(* IEC 61131-3 sources: AXOpen/src/components.rexroth.drives/ctrl/src/AxoIndraDrive (part 3) *)

            Valid			:= 	MC_ReadParameterDone_;
            Busy			:= 	MC_ReadParameterActive_;
            Error			:= 	MC_ReadParameterError_;
            ErrorID			:= 	TO_DINT(MC_ReadParameterErrorID_);
            IF Valid THEN
                Value			:= 	MC_ReadParameterValue_;
            ELSE
                Value			:= 	0;
            END_IF;
        END_METHOD

        ///<summary>
        /// This method returns the value of a vendor specific parameter with datatype REAL.
        ///<summary>
        VAR INTERNAL
            MC_ReadRealParameterEnable_PV		: 	BOOL := FALSE;		//Enable - previous value
            MC_ReadRealParameterDone_PV			:	BOOL := FALSE;		//Done - previous value
            MC_ReadRealParameterCallNumber		: 	INT; 				//Call number of the method MC_ReadRealParameter
            MC_ReadRealParameterNumber_PV		: 	DINT;				//ParameterNumber - previous value (stored at rising edge of the Enable)
            MC_ReadRealParameterFirstCall		: 	BOOL;				//First call of the method MC_ReadRealParameter
            MC_ReadRealParameterDone_			:	BOOL;
            MC_ReadRealParameterActive_			:	BOOL := FALSE;
            MC_ReadRealParameterError_			:	BOOL;
            MC_ReadRealParameterErrorID_		:	eAxoIndraDriveErrorCode;
            MC_ReadRealParameterValue_			:	REAL;
        END_VAR
        METHOD PUBLIC OVERRIDE MC_ReadRealParameter
            VAR_INPUT
                AxisRef         :   AXOpen.Components.Abstractions.Drives.IAxoAxisReference;
                Enable          :   BOOL;                       //  Get the value of the parameter continuously while enabled
                ParameterNumber :   DINT;                       //  Number of the parameter. One can also use symbolic parameter names which are declared as VAR CONST.
            END_VAR
            VAR_OUTPUT
                Valid           :   BOOL;                       //  A valid output is available at the method
                Busy            :   BOOL;                       //  The method is not finished and new output values are to be expected
                Error           :   BOOL;                       //  Signals that an error has occurred within the method
                ErrorID         :   DINT;                       //  Error identification
                Value           :   REAL;                       //  Value of the specified parameter in the datatype, as specified by the vendor
            END_VAR
            VAR
                _AxisReference :  REF_TO AXOpen.Components.Rexroth.Drives.AxoIndraDriveAxisReference;
                Dummy : BOOL;
            END_VAR

            _AxisReference ?= AxisRef;

            Messenger.ActivateOnCondition(ULINT#1413,_AxisReference = NULL, eAxoMessageCategory#ProgrammingError);

            IF(_AxisReference = NULL) THEN
                RETURN;
            END_IF;

            IF Enable THEN
                MC_ReadRealParameterFirstCall := TRUE;
                IF _AxisReference^.Data.CheckAccessOK THEN
                    IF Enable AND NOT MC_ReadRealParameterEnable_PV THEN(*	raising edge of Enable *)
                        IF NOT _AxisReference^.Data.ActiveAcyclicCommunication THEN
                            _AxisReference^.Data.CallNumberAcyclic := _AxisReference^.Data.CallNumberAcyclic + INT#2;
                            MC_ReadRealParameterCallNumber := _AxisReference^.Data.CallNumberAcyclic;
                            MC_ReadRealParameterNumber_PV := ParameterNumber;
                            _AxisReference^.Data.WriteParameter := FALSE;
                            _AxisReference^.Data.SelectDataType := UINT#2;
                            _AxisReference^.Data.ParameterNumber := MC_ReadRealParameterNumber_PV;
                            MC_ReadRealParameterError_ := FALSE;
                            MC_ReadRealParameterErrorID_ := AXOpen.Components.Rexroth.Drives.eAxoIndraDriveErrorCode#NONE_ERROR;
                        ELSE
                            MC_ReadRealParameterError_ := TRUE;
                            MC_ReadRealParameterErrorID_ := AXOpen.Components.Rexroth.Drives.eAxoIndraDriveErrorCode#ACCESS_ERROR;
                        END_IF;
                    END_IF;
                ELSE
                    MC_ReadRealParameterCallNumber := MC_ReadRealParameterCallNumber - INT#1;
                    MC_ReadRealParameterError_ := TRUE;
                    MC_ReadRealParameterErrorID_ := AXOpen.Components.Rexroth.Drives.eAxoIndraDriveErrorCode#RESOURCE_ERROR;
                END_IF;
            END_IF;
            IF MC_ReadRealParameterFirstCall THEN
                IF MC_ReadRealParameterCallNumber = _AxisReference^.Data.CallNumberAcyclic AND Enable	THEN
                    _AxisReference^.Data.CallAxisParameterMethod := TRUE;
                    _AxisReference^.Data.EnableAcyclicCommunication := TRUE;
                    THIS.AcyclicCommunicationCall(AxisRef :=  _AxisReference , DPV1ParameterNumber := TRUE, Active => Dummy);
                    Busy := _AxisReference^.Data.ActiveAcyclicCommunication;
                    IF _AxisReference^.Data.DoneAcyclicCommunication THEN
                        MC_ReadRealParameterDone_ := TRUE;
                        MC_ReadRealParameterActive_ := FALSE;
                        MC_ReadRealParameterValue_ := _AxisReference^.Data.ReadValueReal;
                    END_IF;
                    IF _AxisReference^.Data.Error_AcyclicCommunication THEN
                        MC_ReadRealParameterCallNumber := MC_ReadRealParameterCallNumber - INT#1;
                        MC_ReadRealParameterDone_ := FALSE;
                        MC_ReadRealParameterActive_ := FALSE;
                        MC_ReadRealParameterError_ := _AxisReference^.Data.Error_AcyclicCommunication;
                        MC_ReadRealParameterErrorID_ := _AxisReference^.Data.ErrorID_AcyclicCommunication;
                        _AxisReference^.Data.CallAxisParameterMethod := TRUE;
                        _AxisReference^.Data.EnableAcyclicCommunication := FALSE;
                        THIS.AcyclicCommunicationCall(AxisRef :=  _AxisReference , DPV1ParameterNumber := TRUE, Active => Dummy);
                    ELSIF  _AxisReference^.Data.CallAxisParameterMethod THEN
                        MC_ReadRealParameterCallNumber := MC_ReadRealParameterCallNumber - INT#1;
                        MC_ReadRealParameterDone_ := FALSE;
                        MC_ReadRealParameterActive_ := FALSE;
                        MC_ReadRealParameterError_ := TRUE;
                        MC_ReadRealParameterErrorID_ := AXOpen.Components.Rexroth.Drives.eAxoIndraDriveErrorCode#RESOURCE_ERROR;
                        _AxisReference^.Data.EnableAcyclicCommunication := FALSE;
                    END_IF;
                ELSIF Enable AND MC_ReadRealParameterEnable_PV AND MC_ReadRealParameterCallNumber = _AxisReference^.Data.CallNumberAcyclic THEN
                    _AxisReference^.Data.CallAxisParameterMethod := TRUE;
                    _AxisReference^.Data.EnableAcyclicCommunication := FALSE;
                    THIS.AcyclicCommunicationCall(AxisRef :=  _AxisReference , DPV1ParameterNumber := TRUE, Active => Dummy);
                    MC_ReadRealParameterDone_ := FALSE;
                    MC_ReadRealParameterActive_ := FALSE;
                    MC_ReadRealParameterValue_ := 0;
                    MC_ReadRealParameterError_ := FALSE;
                    MC_ReadRealParameterErrorID_ := AXOpen.Components.Rexroth.Drives.eAxoIndraDriveErrorCode#NONE_ERROR;
                ELSIF NOT Enable AND MC_ReadRealParameterEnable_PV THEN
                    MC_ReadRealParameterDone_ := FALSE;
                    MC_ReadRealParameterActive_ := FALSE;
                    MC_ReadRealParameterValue_ := 0;
                    MC_ReadRealParameterError_ := FALSE;
                    MC_ReadRealParameterErrorID_ := AXOpen.Components.Rexroth.Drives.eAxoIndraDriveErrorCode#NONE_ERROR;
                    _AxisReference^.Data.ActiveAcyclicCommunication := FALSE;
                    _AxisReference^.Data.DoneAcyclicCommunication := FALSE;
                END_IF;
            END_IF;
            MC_ReadRealParameterEnable_PV := Enable;

            Valid			:= 	MC_ReadRealParameterDone_;
            Busy			:= 	MC_ReadRealParameterActive_;
            Error			:= 	MC_ReadRealParameterError_;
            ErrorID			:= 	TO_DINT(MC_ReadRealParameterErrorID_);
            IF Valid THEN
                Value			:= 	MC_ReadRealParameterValue_;
            ELSE
                Value			:= 	0;
            END_IF;
        END_METHOD

        ///<summary>
        /// This method returns the value of a vendor specific parameter with datatype BOOL.
        ///<summary>
        METHOD PUBLIC OVERRIDE MC_ReadBoolParameter
            VAR_INPUT
                AxisRef         :   AXOpen.Components.Abstractions.Drives.IAxoAxisReference;
                Enable          :   BOOL;                       //  Get the value of the parameter continuously while enabled
                ParameterNumber :   DINT;                       //  Number of the parameter. One can also use symbolic parameter names which are declared as VAR CONST.
            END_VAR
            VAR_OUTPUT
                Valid           :   BOOL;                       //  A valid output is available at the method
                Busy            :   BOOL;                       //  The method is not finished and new output values are to be expected
                Error           :   BOOL;                       //  Signals that an error has occurred within the method
                ErrorID         :   DINT;                       //  Error identification
                Value           :   BOOL;                       //  Value of the specified parameter in the datatype, as specified by the vendor
            END_VAR
            VAR
                _AxisReference :  REF_TO AXOpen.Components.Rexroth.Drives.AxoIndraDriveAxisReference;
                Dummy : BOOL;
            END_VAR
            RETURN;

            _AxisReference ?= AxisRef;

            Messenger.ActivateOnCondition(ULINT#1414,_AxisReference = NULL, eAxoMessageCategory#ProgrammingError);

            IF(_AxisReference = NULL) THEN
                RETURN;
            END_IF;

        END_METHOD

        ///<summary>
        /// This method modifies the value of a vendor specific parameter.
        ///<summary>
        VAR INTERNAL
            MC_WriteParameterExecute_PV			: 	BOOL := FALSE;		//Execute - previous value
            MC_WriteParameterDone_PV			:	BOOL := FALSE;		//Done - previous value
            MC_WriteParameterCallNumber			: 	DINT; 				//Call number of the method MC_WriteParameter
            MC_WriteParameterFirstCall			: 	BOOL;				//First call of the method MC_WriteParameter
            MC_WriteParameterDone_				:	BOOL;
            MC_WriteParameterActive_			:	BOOL := FALSE;
            MC_WriteParameterError_				:	BOOL;
            MC_WriteParameterErrorID_			:	eAxoIndraDriveErrorCode;
        END_VAR
        METHOD PUBLIC OVERRIDE MC_WriteParameter
            VAR_INPUT
                AxisRef         :   AXOpen.Components.Abstractions.Drives.IAxoAxisReference;
                Execute         :   BOOL;                       //  Write the value of the parameter at rising edge
                ParameterNumber :   DINT;                       //  Number of the parameter (correspondence between number andparameter is specified in the table above)
                Value           :   LINT;                       //  New value of the specified parameter
                ExecutionMode   :   AXOpen.Components.Abstractions.Drives.eAxoExecutionMode;          //  Defines the chronological sequence of the method.
            END_VAR
            VAR_OUTPUT
                Done            :   BOOL;                       //  Parameter successfully written
                Busy            :   BOOL;                       //  The method is not finished and new output values are to be expected.
                Error           :   BOOL;                       //  Signals that an error has occurred within the method
                ErrorID         :   DINT;                       //  Error identification
            END_VAR
            VAR
                _AxisReference :  REF_TO AXOpen.Components.Rexroth.Drives.AxoIndraDriveAxisReference;
                Dummy : BOOL;
            END_VAR

            _AxisReference ?= AxisRef;

            Messenger.ActivateOnCondition(ULINT#1415,_AxisReference = NULL, eAxoMessageCategory#ProgrammingError);

            IF(_AxisReference = NULL) THEN
                RETURN;
            END_IF;

            IF Execute THEN
                MC_WriteParameterFirstCall := TRUE;
                IF _AxisReference^.Data.CheckAccessOK THEN
                    IF Execute AND NOT MC_WriteParameterExecute_PV THEN(*	raising edge of Execute *)
                        IF NOT _AxisReference^.Data.ActiveAcyclicCommunication THEN
                            _AxisReference^.Data.CallNumberAcyclic := _AxisReference^.Data.CallNumberAcyclic + INT#2;
                            MC_WriteParameterCallNumber := _AxisReference^.Data.CallNumberAcyclic;
                            _AxisReference^.Data.WriteParameter := TRUE;
                            _AxisReference^.Data.SelectDataType := UINT#1;
                            _AxisReference^.Data.ParameterNumber := ParameterNumber;
                            _AxisReference^.Data.WriteValueLint := Value;
                            MC_WriteParameterError_ := FALSE;
                            MC_WriteParameterErrorID_ := AXOpen.Components.Rexroth.Drives.eAxoIndraDriveErrorCode#NONE_ERROR;
                        ELSE
                            MC_WriteParameterError_ := TRUE;
                            MC_WriteParameterErrorID_ := AXOpen.Components.Rexroth.Drives.eAxoIndraDriveErrorCode#ACCESS_ERROR;
                        END_IF;
                    END_IF;
                ELSE
                    MC_WriteParameterCallNumber := MC_WriteParameterCallNumber - INT#1;
                    MC_WriteParameterError_ := TRUE;
                    MC_WriteParameterErrorID_ := AXOpen.Components.Rexroth.Drives.eAxoIndraDriveErrorCode#RESOURCE_ERROR;
                END_IF;
            END_IF;
            IF MC_WriteParameterFirstCall THEN
                IF MC_WriteParameterCallNumber = _AxisReference^.Data.CallNumberAcyclic AND Execute THEN
                    _AxisReference^.Data.CallAxisParameterMethod := TRUE;
                    _AxisReference^.Data.EnableAcyclicCommunication := TRUE;
                    THIS.AcyclicCommunicationCall(AxisRef := _AxisReference , DPV1ParameterNumber := TRUE, Active => Dummy);
                    MC_WriteParameterActive_ := _AxisReference^.Data.ActiveAcyclicCommunication;
                    IF _AxisReference^.Data.DoneAcyclicCommunication THEN
                        MC_WriteParameterCallNumber := MC_WriteParameterCallNumber - INT#1;
                        MC_WriteParameterDone_ := TRUE;
                        MC_WriteParameterActive_ := FALSE;
                    END_IF;
                    IF _AxisReference^.Data.Error_AcyclicCommunication THEN
                        MC_WriteParameterCallNumber := MC_WriteParameterCallNumber - INT#1;
                        MC_WriteParameterDone_ := FALSE;
                        MC_WriteParameterActive_ := FALSE;
                        MC_WriteParameterError_ := _AxisReference^.Data.Error_AcyclicCommunication;
                        MC_WriteParameterErrorID_ := _AxisReference^.Data.ErrorID_AcyclicCommunication;
                        _AxisReference^.Data.CallAxisParameterMethod := TRUE;
                        _AxisReference^.Data.EnableAcyclicCommunication := FALSE;
                        THIS.AcyclicCommunicationCall(AxisRef := _AxisReference , DPV1ParameterNumber := TRUE, Active => Dummy);
                    ELSIF _AxisReference^.Data.CallAxisParameterMethod THEN
                        MC_WriteParameterCallNumber := MC_WriteParameterCallNumber - INT#1;
                        MC_WriteParameterDone_ := FALSE;
                        MC_WriteParameterActive_ := FALSE;
                        MC_WriteParameterError_ := TRUE;
                        MC_WriteParameterErrorID_ := AXOpen.Components.Rexroth.Drives.eAxoIndraDriveErrorCode#RESOURCE_ERROR;
                        _AxisReference^.Data.EnableAcyclicCommunication := FALSE;
                    END_IF;
                ELSIF NOT Execute AND NOT MC_WriteParameterExecute_PV AND MC_WriteParameterCallNumber = _AxisReference^.Data.CallNumberAcyclic THEN
                    _AxisReference^.Data.CallAxisParameterMethod := TRUE;
                    _AxisReference^.Data.EnableAcyclicCommunication := FALSE;
                    THIS.AcyclicCommunicationCall(AxisRef := _AxisReference , DPV1ParameterNumber := TRUE, Active => Dummy);
                    MC_WriteParameterDone_ := FALSE;
                    MC_WriteParameterActive_ := FALSE;
                    MC_WriteParameterError_ := FALSE;
                    MC_WriteParameterErrorID_ := AXOpen.Components.Rexroth.Drives.eAxoIndraDriveErrorCode#NONE_ERROR;
                ELSIF NOT Execute AND MC_WriteParameterExecute_PV THEN
                    MC_WriteParameterDone_ := FALSE;
                    MC_WriteParameterActive_ := FALSE;
                    MC_WriteParameterError_ := FALSE;
                    MC_WriteParameterErrorID_ := AXOpen.Components.Rexroth.Drives.eAxoIndraDriveErrorCode#NONE_ERROR;
                END_IF;
            END_IF;
            MC_WriteParameterExecute_PV := Execute;

            Done		:= MC_WriteParameterDone_;
            Busy 		:= MC_WriteParameterActive_;
            Error 		:= MC_WriteParameterError_;
            ErrorID 	:= TO_DINT(MC_WriteParameterErrorID_);
        END_METHOD

        ///<summary>
        /// This method modifies the value of a vendor specific parameter of type Real.
        ///<summary>
        VAR INTERNAL
            MC_WriteRealParameterExecute_PV		: 	BOOL := FALSE;		//Execute - previous value
            MC_WriteRealParameterDone_PV		:	BOOL := FALSE;		//Done - previous value
            MC_WriteRealParameterCallNumber		: 	INT; 				//Call number of the method MC_WriteRealParameter
            MC_WriteRealParameterFirstCall		: 	BOOL;				//First call of the method MC_WriteRealParameter
            MC_WriteRealParameterDone_			:	BOOL;
            MC_WriteRealParameterActive_		:	BOOL := FALSE;
            MC_WriteRealParameterError_			:	BOOL;
            MC_WriteRealParameterErrorID_		:	eAxoIndraDriveErrorCode;
        END_VAR
        METHOD PUBLIC OVERRIDE MC_WriteRealParameter
            VAR_INPUT
                AxisRef         :   AXOpen.Components.Abstractions.Drives.IAxoAxisReference;
                Execute         :   BOOL;                       //  Write the value of the parameter at rising edge
                ParameterNumber :   DINT;                       //  Number of the parameter (correspondence between number andparameter is specified in the table above)
                Value           :   REAL;                       //  New value of the specified parameter
                ExecutionMode   :   AXOpen.Components.Abstractions.Drives.eAxoExecutionMode;          //  Defines the chronological sequence of the method.
            END_VAR
            VAR_OUTPUT
                Done            :   BOOL;                       //  Parameter successfully written
                Busy            :   BOOL;                       //  The method is not finished and new output values are to be expected.
                Error           :   BOOL;                       //  Signals that an error has occurred within the method
                ErrorID         :   DINT;                       //  Error identification
            END_VAR
            VAR
                _AxisReference :  REF_TO AXOpen.Components.Rexroth.Drives.AxoIndraDriveAxisReference;
                Dummy : BOOL;
            END_VAR

            _AxisReference ?= AxisRef;

            Messenger.ActivateOnCondition(ULINT#1416,_AxisReference = NULL, eAxoMessageCategory#ProgrammingError);

            IF(_AxisReference = NULL) THEN
                RETURN;
            END_IF;

            IF Execute THEN
                MC_WriteRealParameterFirstCall := TRUE;
                IF _AxisReference^.Data.CheckAccessOK THEN
                    IF Execute AND NOT MC_WriteRealParameterExecute_PV THEN (*	raising edge of Execute *)
                        IF NOT _AxisReference^.Data.ActiveAcyclicCommunication THEN
                            _AxisReference^.Data.CallNumberAcyclic := _AxisReference^.Data.CallNumberAcyclic + INT#2;
                            MC_WriteRealParameterCallNumber := _AxisReference^.Data.CallNumberAcyclic;
                            _AxisReference^.Data.WriteParameter := TRUE;
                            _AxisReference^.Data.SelectDataType := UINT#2;
                            _AxisReference^.Data.ParameterNumber := ParameterNumber;
                            _AxisReference^.Data.WriteValueReal := Value;
                            MC_WriteRealParameterError_ := FALSE;
                            MC_WriteRealParameterErrorID_ := AXOpen.Components.Rexroth.Drives.eAxoIndraDriveErrorCode#NONE_ERROR;
                        ELSE
                            MC_WriteRealParameterError_ := TRUE;
                            MC_WriteRealParameterErrorID_ := AXOpen.Components.Rexroth.Drives.eAxoIndraDriveErrorCode#ACCESS_ERROR;
                        END_IF;
                    END_IF;
                ELSE
                    MC_WriteRealParameterCallNumber := MC_WriteRealParameterCallNumber - INT#1;
                    MC_WriteRealParameterError_ := TRUE;
                    MC_WriteRealParameterErrorID_ := AXOpen.Components.Rexroth.Drives.eAxoIndraDriveErrorCode#RESOURCE_ERROR;
                END_IF;
            END_IF;
            IF MC_WriteRealParameterFirstCall THEN
                IF MC_WriteRealParameterCallNumber = _AxisReference^.Data.CallNumberAcyclic AND Execute THEN
                    _AxisReference^.Data.CallAxisParameterMethod := TRUE;
                    _AxisReference^.Data.EnableAcyclicCommunication := TRUE;
                    THIS.AcyclicCommunicationCall(AxisRef := _AxisReference , DPV1ParameterNumber := TRUE, Active => Dummy);
                    MC_WriteRealParameterActive_ := _AxisReference^.Data.ActiveAcyclicCommunication;
                    IF _AxisReference^.Data.DoneAcyclicCommunication THEN
                        MC_WriteRealParameterCallNumber := MC_WriteRealParameterCallNumber - INT#1;
                        MC_WriteRealParameterDone_ := TRUE;
                        MC_WriteRealParameterActive_ := FALSE;
                    END_IF;
                    IF _AxisReference^.Data.Error_AcyclicCommunication THEN
                        MC_WriteRealParameterCallNumber := MC_WriteRealParameterCallNumber - INT#1;
                        MC_WriteRealParameterDone_ := FALSE;
                        MC_WriteRealParameterActive_ := FALSE;
                        MC_WriteRealParameterError_ := _AxisReference^.Data.Error_AcyclicCommunication;
                        MC_WriteRealParameterErrorID_ := _AxisReference^.Data.ErrorID_AcyclicCommunication;
                        _AxisReference^.Data.CallAxisParameterMethod := TRUE;
                        _AxisReference^.Data.EnableAcyclicCommunication := FALSE;
                        THIS.AcyclicCommunicationCall(AxisRef := _AxisReference , DPV1ParameterNumber := TRUE, Active => Dummy);
                    ELSIF  _AxisReference^.Data.CallAxisParameterMethod THEN
                        MC_WriteRealParameterCallNumber := MC_WriteRealParameterCallNumber - INT#1;
                        MC_WriteRealParameterDone_ := FALSE;
                        MC_WriteRealParameterActive_ := FALSE;
                        MC_WriteRealParameterError_ := TRUE;
                        MC_WriteRealParameterErrorID_ := AXOpen.Components.Rexroth.Drives.eAxoIndraDriveErrorCode#RESOURCE_ERROR;
                        _AxisReference^.Data.EnableAcyclicCommunication := FALSE;
                    END_IF;
                ELSIF NOT Execute AND MC_WriteRealParameterExecute_PV AND MC_WriteRealParameterCallNumber = _AxisReference^.Data.CallNumberAcyclic THEN
                    _AxisReference^.Data.CallAxisParameterMethod := TRUE;
                    _AxisReference^.Data.EnableAcyclicCommunication := FALSE;
                    THIS.AcyclicCommunicationCall(AxisRef := _AxisReference , DPV1ParameterNumber := TRUE, Active => Dummy);
                    MC_WriteRealParameterDone_ := FALSE;
                    MC_WriteRealParameterActive_ := FALSE;
                    MC_WriteRealParameterError_ := FALSE;
                    MC_WriteRealParameterErrorID_ := AXOpen.Components.Rexroth.Drives.eAxoIndraDriveErrorCode#NONE_ERROR;
                ELSIF NOT Execute AND MC_WriteRealParameterExecute_PV THEN
                    MC_WriteRealParameterDone_ := FALSE;
                    MC_WriteRealParameterActive_ := FALSE;
                    MC_WriteRealParameterError_ := FALSE;
                    MC_WriteRealParameterErrorID_ := AXOpen.Components.Rexroth.Drives.eAxoIndraDriveErrorCode#NONE_ERROR;
                END_IF;
            END_IF;
            MC_WriteRealParameterExecute_PV := Execute;

            Done			:= MC_WriteRealParameterDone_;
            Busy			:= MC_WriteRealParameterActive_;
            Error			:= MC_WriteRealParameterError_;
            ErrorID			:= TO_DINT(MC_WriteRealParameterErrorID_);
        END_METHOD

        ///<summary>
        /// This method modifies the value of a vendor specific parameter of type BOOL.
        ///<summary>
        METHOD PUBLIC OVERRIDE MC_WriteBoolParameter
            VAR_INPUT
                AxisRef         :   AXOpen.Components.Abstractions.Drives.IAxoAxisReference;
                Execute         :   BOOL;                       //  Write the value of the parameter at rising edge
                ParameterNumber :   DINT;                       //  Number of the parameter (correspondence between number andparameter is specified in the table above)
                Value           :   BOOL;                       //  New value of the specified parameter
                ExecutionMode   :   AXOpen.Components.Abstractions.Drives.eAxoExecutionMode;          //  Defines the chronological sequence of the method.
            END_VAR
            VAR_OUTPUT
                Done            :   BOOL;                       //  Parameter successfully written
                Busy            :   BOOL;                       //  The method is not finished and new output values are to be expected.
                Error           :   BOOL;                       //  Signals that an error has occurred within the method
                ErrorID         :   DINT;                       //  Error identification
            END_VAR
            VAR
                _AxisReference :  REF_TO AXOpen.Components.Rexroth.Drives.AxoIndraDriveAxisReference;
                Dummy : BOOL;
            END_VAR

            _AxisReference ?= AxisRef;

            Messenger.ActivateOnCondition(ULINT#1417,_AxisReference = NULL, eAxoMessageCategory#ProgrammingError);

            IF(_AxisReference = NULL) THEN
                RETURN;
            END_IF;

        END_METHOD

        ///<summary>
        /// This method gives access to the value of the input, referenced by the datatype MC_INPUT_REF.
        /// It provides the value of the referenced input (BOOL).
        ///<summary>
        VAR INTERNAL
            MC_ReadDigitalInputEnable_PV		: 	BOOL := FALSE;		//Enable - previous value
            MC_ReadDigitalInputDone_PV			:	BOOL := FALSE;		//Done - previous value
            MC_ReadDigitalInputCallNumber		: 	INT; 				//Call number of the method MC_ReadDigitalInput
            MC_ReadDigitalInputNumber_PV		: 	DINT;				//DigitalInputNumber - previous value (stored at rising edge of the Enable)
            MC_ReadDigitalInputFirstCall		: 	BOOL;				//First call of the method MC_ReadDigitalInput
            MC_ReadDigitalInputDone_			:	BOOL;
            MC_ReadDigitalInputActive_			:	BOOL := FALSE;
            MC_ReadDigitalInputError_			:	BOOL;
            MC_ReadDigitalInputErrorID_			:	eAxoIndraDriveErrorCode;
            MC_ReadDigitalInputValue_			:	DINT;
        END_VAR
        METHOD PUBLIC OVERRIDE MC_ReadDigitalInput
            VAR_INPUT
                AxisRef         :   AXOpen.Components.Abstractions.Drives.IAxoAxisReference;
                Enable          :   BOOL;                       //  Get the value of the selected input signal continuously while enabled
                InputNumber     :   INT;                        //  Selects the input. Can be part of MC_INPUT_REF, if only one single input is referenced.
            END_VAR
            VAR_OUTPUT
                Valid           :   BOOL;                       //  A valid output is available at the method
                Busy            :   BOOL;                       //  The method is not finished and new output values are to be expected
                Error           :   BOOL;                       //  Signals that an error has occurred within the method
                ErrorID         :   DINT;                       //  Error identification
                Value           :   BOOL;                       //  The value of the selected input signal
            END_VAR
            VAR
                _AxisReference :  REF_TO AXOpen.Components.Rexroth.Drives.AxoIndraDriveAxisReference;
                Dummy : BOOL;
            END_VAR

            _AxisReference ?= AxisRef;

            Messenger.ActivateOnCondition(ULINT#1418,_AxisReference = NULL, eAxoMessageCategory#ProgrammingError);

            IF(_AxisReference = NULL) THEN
                RETURN;
            END_IF;

            IF Enable THEN
                MC_ReadDigitalInputFirstCall := TRUE;
                IF _AxisReference^.Data.CheckAccessOK THEN
                    IF Enable AND NOT MC_ReadDigitalInputEnable_PV THEN(*	raising edge of Enable *)
                        IF NOT _AxisReference^.Data.ActiveAcyclicCommunication THEN
                            _AxisReference^.Data.CallNumberAcyclic := _AxisReference^.Data.CallNumberAcyclic + INT#2;
                            MC_ReadDigitalInputCallNumber := _AxisReference^.Data.CallNumberAcyclic;
                            MC_ReadDigitalInputNumber_PV := DINT#33071;
                            _AxisReference^.Data.WriteParameter := FALSE;
                            _AxisReference^.Data.SelectDataType := UINT#1;
                            _AxisReference^.Data.ParameterNumber := MC_ReadDigitalInputNumber_PV;
                            MC_ReadDigitalInputError_ := FALSE;
                            MC_ReadDigitalInputErrorID_ := AXOpen.Components.Rexroth.Drives.eAxoIndraDriveErrorCode#NONE_ERROR;
                        ELSE
                            MC_ReadDigitalInputError_ := TRUE;
                            MC_ReadDigitalInputErrorID_ := AXOpen.Components.Rexroth.Drives.eAxoIndraDriveErrorCode#ACCESS_ERROR;
                        END_IF;
                    END_IF;
                ELSE
                    MC_ReadDigitalInputCallNumber := MC_ReadDigitalInputCallNumber - INT#1;
                    MC_ReadDigitalInputError_ := TRUE;
                    MC_ReadDigitalInputErrorID_ := AXOpen.Components.Rexroth.Drives.eAxoIndraDriveErrorCode#RESOURCE_ERROR;
                END_IF;
            END_IF;
            IF MC_ReadDigitalInputFirstCall THEN
                IF MC_ReadDigitalInputCallNumber = _AxisReference^.Data.CallNumberAcyclic AND Enable	THEN
                    _AxisReference^.Data.CallAxisParameterMethod := TRUE;
                    _AxisReference^.Data.EnableAcyclicCommunication := TRUE;
                    THIS.AcyclicCommunicationCall(AxisRef :=  _AxisReference , DPV1ParameterNumber := TRUE, Active => Dummy);
                    Busy := _AxisReference^.Data.ActiveAcyclicCommunication;
                    IF _AxisReference^.Data.DoneAcyclicCommunication THEN
                        MC_ReadDigitalInputDone_ := TRUE;
                        MC_ReadDigitalInputActive_ := FALSE;
                        MC_ReadDigitalInputValue_ := _AxisReference^.Data.ReadValueDint;
                    END_IF;
                    IF _AxisReference^.Data.Error_AcyclicCommunication THEN
                        MC_ReadDigitalInputCallNumber := MC_ReadDigitalInputCallNumber - INT#1;
                        MC_ReadDigitalInputDone_ := FALSE;
                        MC_ReadDigitalInputActive_ := FALSE;
                        MC_ReadDigitalInputError_ := _AxisReference^.Data.Error_AcyclicCommunication;
                        MC_ReadDigitalInputErrorID_ := _AxisReference^.Data.ErrorID_AcyclicCommunication;
                        _AxisReference^.Data.CallAxisParameterMethod := TRUE;
                        _AxisReference^.Data.EnableAcyclicCommunication := FALSE;
                        THIS.AcyclicCommunicationCall(AxisRef :=  _AxisReference , DPV1ParameterNumber := TRUE, Active => Dummy);
                    ELSIF  _AxisReference^.Data.CallAxisParameterMethod THEN
                        MC_ReadDigitalInputCallNumber := MC_ReadDigitalInputCallNumber - INT#1;
                        MC_ReadDigitalInputDone_ := FALSE;
                        MC_ReadDigitalInputActive_ := FALSE;
                        MC_ReadDigitalInputError_ := TRUE;
                        MC_ReadDigitalInputErrorID_ := AXOpen.Components.Rexroth.Drives.eAxoIndraDriveErrorCode#RESOURCE_ERROR;
                        _AxisReference^.Data.EnableAcyclicCommunication := FALSE;
                    END_IF;
                ELSIF Enable AND MC_ReadDigitalInputEnable_PV AND MC_ReadDigitalInputCallNumber = _AxisReference^.Data.CallNumberAcyclic THEN
                    _AxisReference^.Data.CallAxisParameterMethod := TRUE;
                    _AxisReference^.Data.EnableAcyclicCommunication := FALSE;
                    THIS.AcyclicCommunicationCall(AxisRef :=  _AxisReference , DPV1ParameterNumber := TRUE, Active => Dummy);
                    MC_ReadDigitalInputDone_ := FALSE;
                    MC_ReadDigitalInputActive_ := FALSE;
                    MC_ReadDigitalInputValue_ := DINT#0;
                    MC_ReadDigitalInputError_ := FALSE;
                    MC_ReadDigitalInputErrorID_ := AXOpen.Components.Rexroth.Drives.eAxoIndraDriveErrorCode#NONE_ERROR;
                ELSIF NOT Enable AND MC_ReadDigitalInputEnable_PV THEN
                    MC_ReadDigitalInputDone_ := FALSE;
                    MC_ReadDigitalInputActive_ := FALSE;
                    MC_ReadDigitalInputValue_ := DINT#0;
                    MC_ReadDigitalInputError_ := FALSE;
                    MC_ReadDigitalInputErrorID_ := AXOpen.Components.Rexroth.Drives.eAxoIndraDriveErrorCode#NONE_ERROR;
                    _AxisReference^.Data.ActiveAcyclicCommunication := FALSE;
                    _AxisReference^.Data.DoneAcyclicCommunication := FALSE;
                END_IF;
            END_IF;
            MC_ReadDigitalInputEnable_PV := Enable;

            Valid			:= 	MC_ReadDigitalInputDone_;
            Busy			:= 	MC_ReadDigitalInputActive_;
            Error			:= 	MC_ReadDigitalInputError_;
            ErrorID			:= 	TO_DINT(MC_ReadDigitalInputErrorID_);

            IF Valid THEN
                IF InputNumber >=0 AND InputNumber <=15 THEN
                    Value			:= 	System.BitAccess.GetBit(TO_DWORD(MC_ReadDigitalInputValue_),TO_USINT(InputNumber));
                END_IF;
            ELSE
                Value			:= 	FALSE;
            END_IF;
        END_METHOD

        ///<summary>
        /// This method provides access to the value of a digital output, referenced by the datatype MC_OUTPUT_REF.
        /// It provides the value of the referenced output (BOOL).
        ///<summary>
        VAR INTERNAL
            MC_ReadDigitalOutputEnable_PV		: 	BOOL := FALSE;		//Enable - previous value
            MC_ReadDigitalOutputDone_PV			:	BOOL := FALSE;		//Done - previous value
            MC_ReadDigitalOutputCallNumber		: 	INT; 				//Call number of the method MC_ReadDigitalOutput
            MC_ReadDigitalOutputNumber_PV		: 	DINT;				//DigitalIOutputNumber - previous value (stored at rising edge of the Enable)
            MC_ReadDigitalOutputFirstCall		: 	BOOL;				//First call of the method MC_ReadDigitalOutput
            MC_ReadDigitalOutputDone_			:	BOOL;
            MC_ReadDigitalOutputActive_			:	BOOL := FALSE;
            MC_ReadDigitalOutputError_			:	BOOL;
            MC_ReadDigitalOutputErrorID_		:	eAxoIndraDriveErrorCode;
            MC_ReadDigitalOutputValue_			:	DINT;
        END_VAR
        METHOD PUBLIC OVERRIDE MC_ReadDigitalOutput
            VAR_INPUT
                AxisRef         :   AXOpen.Components.Abstractions.Drives.IAxoAxisReference;
                Enable          :   BOOL;                       //  Get the value of the selected output signal continuously while enabled
                OutputNumber    :   INT;                        //  Selects the output. Can be part of MC_OUTPUT_REF, if only one single output is referenced.
            END_VAR
            VAR_OUTPUT
                Valid           :   BOOL;                       //  A valid output is available at the method
                Busy            :   BOOL;                       //  The method is not finished and new output values are to be expected
                Error           :   BOOL;                       //  Signals that an error has occurred within the method
                ErrorID         :   DINT;                       //  Error identification
                Value           :   BOOL;                       //  The value of the selected output signal
            END_VAR
            VAR
                _AxisReference :  REF_TO AXOpen.Components.Rexroth.Drives.AxoIndraDriveAxisReference;
                Dummy : BOOL;
            END_VAR

            _AxisReference ?= AxisRef;

            Messenger.ActivateOnCondition(ULINT#1419,_AxisReference = NULL, eAxoMessageCategory#ProgrammingError);

            IF(_AxisReference = NULL) THEN
                RETURN;
            END_IF;

            IF Enable THEN
                MC_ReadDigitalOutputFirstCall := TRUE;
                IF _AxisReference^.Data.CheckAccessOK THEN
                    IF Enable AND NOT MC_ReadDigitalOutputEnable_PV THEN(*	raising edge of Enable *)
                        IF NOT _AxisReference^.Data.ActiveAcyclicCommunication THEN
                            _AxisReference^.Data.CallNumberAcyclic := _AxisReference^.Data.CallNumberAcyclic + INT#2;
                            MC_ReadDigitalOutputCallNumber := _AxisReference^.Data.CallNumberAcyclic;
                            MC_ReadDigitalOutputNumber_PV := DINT#33072; (*P-0-0304, Digital outputs, output image device*)
                            _AxisReference^.Data.WriteParameter := FALSE;
                            _AxisReference^.Data.SelectDataType := UINT#1;
                            _AxisReference^.Data.ParameterNumber := MC_ReadDigitalOutputNumber_PV;
                            MC_ReadDigitalOutputError_ := FALSE;
                            MC_ReadDigitalOutputErrorID_ := AXOpen.Components.Rexroth.Drives.eAxoIndraDriveErrorCode#NONE_ERROR;
                        ELSE
                            MC_ReadDigitalOutputError_ := TRUE;
                            MC_ReadDigitalOutputErrorID_ := AXOpen.Components.Rexroth.Drives.eAxoIndraDriveErrorCode#ACCESS_ERROR;
                        END_IF;
                    END_IF;
                ELSE
                    MC_ReadDigitalOutputCallNumber := MC_ReadDigitalOutputCallNumber - INT#1;
                    MC_ReadDigitalOutputError_ := TRUE;
                    MC_ReadDigitalOutputErrorID_ := AXOpen.Components.Rexroth.Drives.eAxoIndraDriveErrorCode#RESOURCE_ERROR;
                END_IF;
            END_IF;
            IF MC_ReadDigitalOutputFirstCall THEN
                IF MC_ReadDigitalOutputCallNumber = _AxisReference^.Data.CallNumberAcyclic AND Enable	THEN
                    _AxisReference^.Data.CallAxisParameterMethod := TRUE;
                    _AxisReference^.Data.EnableAcyclicCommunication := TRUE;
                    THIS.AcyclicCommunicationCall(AxisRef :=  _AxisReference , DPV1ParameterNumber := TRUE, Active => Dummy);
                    Busy := _AxisReference^.Data.ActiveAcyclicCommunication;
                    IF _AxisReference^.Data.DoneAcyclicCommunication THEN
                        MC_ReadDigitalOutputDone_ := TRUE;
                        MC_ReadDigitalOutputActive_ := FALSE;
                        MC_ReadDigitalOutputValue_ := _AxisReference^.Data.ReadValueDint;
                    END_IF;
                    IF _AxisReference^.Data.Error_AcyclicCommunication THEN
                        MC_ReadDigitalOutputCallNumber := MC_ReadDigitalOutputCallNumber - INT#1;
                        MC_ReadDigitalOutputDone_ := FALSE;
                        MC_ReadDigitalOutputActive_ := FALSE;
                        MC_ReadDigitalOutputError_ := _AxisReference^.Data.Error_AcyclicCommunication;
                        MC_ReadDigitalOutputErrorID_ := _AxisReference^.Data.ErrorID_AcyclicCommunication;
                        _AxisReference^.Data.CallAxisParameterMethod := TRUE;
                        _AxisReference^.Data.EnableAcyclicCommunication := FALSE;
                        THIS.AcyclicCommunicationCall(AxisRef :=  _AxisReference , DPV1ParameterNumber := TRUE, Active => Dummy);
                    ELSIF  _AxisReference^.Data.CallAxisParameterMethod THEN
                        MC_ReadDigitalOutputCallNumber := MC_ReadDigitalOutputCallNumber - INT#1;
                        MC_ReadDigitalOutputDone_ := FALSE;
                        MC_ReadDigitalOutputActive_ := FALSE;
                        MC_ReadDigitalOutputError_ := TRUE;
                        MC_ReadDigitalOutputErrorID_ := AXOpen.Components.Rexroth.Drives.eAxoIndraDriveErrorCode#RESOURCE_ERROR;
                        _AxisReference^.Data.EnableAcyclicCommunication := FALSE;
                    END_IF;
                ELSIF Enable AND MC_ReadDigitalOutputEnable_PV AND MC_ReadDigitalOutputCallNumber = _AxisReference^.Data.CallNumberAcyclic THEN
                    _AxisReference^.Data.CallAxisParameterMethod := TRUE;
                    _AxisReference^.Data.EnableAcyclicCommunication := FALSE;
                    THIS.AcyclicCommunicationCall(AxisRef :=  _AxisReference , DPV1ParameterNumber := TRUE, Active => Dummy);
                    MC_ReadDigitalOutputDone_ := FALSE;
                    MC_ReadDigitalOutputActive_ := FALSE;
                    MC_ReadDigitalOutputValue_ := 0;
                    MC_ReadDigitalOutputError_ := FALSE;
                    MC_ReadDigitalOutputErrorID_ := AXOpen.Components.Rexroth.Drives.eAxoIndraDriveErrorCode#NONE_ERROR;
                ELSIF NOT Enable AND MC_ReadDigitalOutputEnable_PV THEN
                    MC_ReadDigitalOutputDone_ := FALSE;
                    MC_ReadDigitalOutputActive_ := FALSE;
                    MC_ReadDigitalOutputValue_ := 0;
                    MC_ReadDigitalOutputError_ := FALSE;
                    MC_ReadDigitalOutputErrorID_ := AXOpen.Components.Rexroth.Drives.eAxoIndraDriveErrorCode#NONE_ERROR;
                    _AxisReference^.Data.ActiveAcyclicCommunication := FALSE;
                    _AxisReference^.Data.DoneAcyclicCommunication := FALSE;
                END_IF;
            END_IF;
            MC_ReadDigitalOutputEnable_PV := Enable;

            Valid			:= 	MC_ReadDigitalOutputDone_;
            Busy			:= 	MC_ReadDigitalOutputActive_;
            Error			:= 	MC_ReadDigitalOutputError_;
            ErrorID			:= 	TO_DINT(MC_ReadDigitalOutputErrorID_);
            IF Valid THEN
                IF OutputNumber >=0 AND OutputNumber <=15 THEN
                    Value			:= 	System.BitAccess.GetBit(TO_WORD(MC_ReadDigitalOutputValue_),TO_USINT(OutputNumber));
                END_IF;
            ELSE
                Value			:= 	FALSE;
            END_IF;
        END_METHOD

        ///<summary>
        /// This method writes a value to the output referenced by the argument ‘Output’ once (with rising edge of Execute)
        ///<summary>
        VAR INTERNAL
            MC_WriteDigitalOutputExecute_PV			: 	BOOL := FALSE;		//Execute - previous value
            MC_WriteDigitalOutputDone_PV			:	BOOL := FALSE;		//Done - previous value
            MC_WriteDigitalOutputCallNumber			: 	INT; 				//Call number of the method MC_WriteDigitalOutput
            MC_WriteDigitalOutputFirstCall			: 	BOOL;				//First call of the method MC_WriteDigitalOutput
            MC_WriteDigitalOutputDone_				:	BOOL;
            MC_WriteDigitalOutputActive_			:	BOOL := FALSE;
            MC_WriteDigitalOutputError_				:	BOOL;
            MC_WriteDigitalOutputErrorID_			:	eAxoIndraDriveErrorCode;
            MC_WriteDigitalOutputState_				:	UINT;
            MC_WriteDigitalOutputValueRead_ 		:	LINT;
            MC_WriteDigitalOutputValueToWrite_		:	LINT;
        END_VAR
        METHOD PUBLIC OVERRIDE MC_WriteDigitalOutput
            VAR_INPUT
                AxisRef         :   AXOpen.Components.Abstractions.Drives.IAxoAxisReference;
                Execute         :   BOOL;                       //  Write the value of the selected output
                OutputNumber    :   INT;                        //  Selects the output. Can be part of MC_OUTPUT_REF, if only one single output is referenced.
                Value           :   BOOL;                       //  The value of the selected output signal
                ExecutionMode   :   AXOpen.Components.Abstractions.Drives.eAxoExecutionMode;          //  Defines the chronological sequence of the method.
            END_VAR
            VAR_OUTPUT
                Done            :   BOOL;                       //  Writing of the output signal value is done
                Busy            :   BOOL;                       //  The method is not finished and new output values are to be expected.
                Error           :   BOOL;                       //  Signals that an error has occurred within the method
                ErrorID         :   DINT;                       //  Error identification
            END_VAR
            VAR
                _AxisReference :  REF_TO AXOpen.Components.Rexroth.Drives.AxoIndraDriveAxisReference;
                Dummy : BOOL;
                Valid_          :   BOOL;
                Error_          :   BOOL;
                ErrorID_        :   DINT;
            END_VAR

            _AxisReference ?= AxisRef;

            Messenger.ActivateOnCondition(ULINT#1420,_AxisReference = NULL, eAxoMessageCategory#ProgrammingError);

            IF(_AxisReference = NULL) THEN
                RETURN;
            END_IF;

            IF Execute THEN
                IF MC_WriteDigitalOutputState_ = UINT#0 THEN
                    AxoReadParameter_ParameterNumber := DINT#33072;
                    THIS.AxoReadParameter(Enable := TRUE, ParameterNumber := DINT#33072, Valid => Valid_, Error => Error_, ErrorID => ErrorID_,Value =>MC_WriteDigitalOutputValueRead_ );
                    IF Error_ THEN
                        Error := TRUE;
                        ErrorID := ErrorID_;
                    END_IF;
                    IF Valid_ THEN
                        IF OutputNumber >= 0 AND OutputNumber <= 15 THEN
                            MC_WriteDigitalOutputValueToWrite_ := MC_WriteDigitalOutputValueRead_;
                            MC_WriteDigitalOutputValueToWrite_	:= TO_DINT(System.BitAccess.SetBit(TO_DWORD(MC_WriteDigitalOutputValueToWrite_),TO_USINT(OutputNumber),Value));
                            MC_WriteDigitalOutputState_ := MC_WriteDigitalOutputState_ + UINT#10;
                        ELSE
                            MC_WriteDigitalOutputError_ := TRUE;
                            MC_WriteDigitalOutputErrorID_ := AXOpen.Components.Rexroth.Drives.eAxoIndraDriveErrorCode#INPUT_RANGE_ERROR;
                        END_IF;
                    END_IF;
                END_IF;
                IF MC_WriteDigitalOutputState_ = UINT#10 THEN
                    THIS.AxoReadParameter(Enable := FALSE, ParameterNumber := DINT#33072, Valid => Valid_, Error => Error_, ErrorID => ErrorID_,Value =>MC_WriteDigitalOutputValueRead_ );
                    IF NOT Valid_ THEN
                        MC_WriteDigitalOutputState_ := MC_WriteDigitalOutputState_ + UINT#10;
                        RETURN;
                    END_IF;
                END_IF;
                IF MC_WriteDigitalOutputState_ >= UINT#20 THEN
                    MC_WriteDigitalOutputFirstCall := TRUE;
                    IF _AxisReference^.Data.CheckAccessOK THEN
                        IF Execute AND NOT MC_WriteDigitalOutputExecute_PV THEN(*	raising edge of Execute *)
                            IF NOT _AxisReference^.Data.ActiveAcyclicCommunication THEN
                                _AxisReference^.Data.CallNumberAcyclic := _AxisReference^.Data.CallNumberAcyclic + INT#2;
                                MC_WriteDigitalOutputCallNumber := _AxisReference^.Data.CallNumberAcyclic;
                                _AxisReference^.Data.WriteParameter := TRUE;
                                _AxisReference^.Data.SelectDataType := UINT#1;
                                _AxisReference^.Data.ParameterNumber := DINT#33072; (*P-0-0304, Digital outputs, output image device*)
                                _AxisReference^.Data.WriteValueLint := MC_WriteDigitalOutputValueToWrite_;
                                MC_WriteDigitalOutputError_ := FALSE;
                                MC_WriteDigitalOutputErrorID_ := AXOpen.Components.Rexroth.Drives.eAxoIndraDriveErrorCode#NONE_ERROR;
                            ELSE
                                MC_WriteDigitalOutputError_ := TRUE;
                                MC_WriteDigitalOutputErrorID_ := AXOpen.Components.Rexroth.Drives.eAxoIndraDriveErrorCode#ACCESS_ERROR;
                            END_IF;
                        END_IF;
                    ELSE
                        MC_WriteDigitalOutputCallNumber := MC_WriteDigitalOutputCallNumber - INT#1;
                        MC_WriteDigitalOutputError_ := TRUE;
                        MC_WriteDigitalOutputErrorID_ := AXOpen.Components.Rexroth.Drives.eAxoIndraDriveErrorCode#RESOURCE_ERROR;
                    END_IF;
                END_IF;
            ELSE
                MC_WriteDigitalOutputState_     :=  UINT#0;
                MC_WriteDigitalOutputDone_      :=  FALSE;
                MC_WriteDigitalOutputActive_    :=  FALSE;
                MC_WriteDigitalOutputError_     :=  FALSE;
                MC_WriteDigitalOutputErrorID_   :=  WORD#0;
                MC_WriteDigitalOutputExecute_PV :=  FALSE;
            END_IF;
            IF MC_WriteDigitalOutputFirstCall THEN
                IF MC_WriteDigitalOutputState_ >= UINT#20 THEN
                    IF MC_WriteDigitalOutputCallNumber = _AxisReference^.Data.CallNumberAcyclic AND Execute THEN
                        _AxisReference^.Data.CallAxisParameterMethod := TRUE;
                        _AxisReference^.Data.EnableAcyclicCommunication := TRUE;
                        THIS.AcyclicCommunicationCall(AxisRef :=  _AxisReference , DPV1ParameterNumber := TRUE, Active => Dummy);
                        MC_WriteDigitalOutputActive_ := _AxisReference^.Data.ActiveAcyclicCommunication;
                        IF _AxisReference^.Data.DoneAcyclicCommunication THEN
                            MC_WriteDigitalOutputCallNumber := MC_WriteDigitalOutputCallNumber -INT#1;
                            MC_WriteDigitalOutputDone_ := TRUE;
                            MC_WriteDigitalOutputActive_ := FALSE;
                        END_IF;
                        IF _AxisReference^.Data.Error_AcyclicCommunication THEN
                            MC_WriteDigitalOutputCallNumber := MC_WriteDigitalOutputCallNumber -INT#1;
                            MC_WriteDigitalOutputDone_ := FALSE;
                            MC_WriteDigitalOutputActive_ := FALSE;
                            MC_WriteDigitalOutputError_ := _AxisReference^.Data.Error_AcyclicCommunication;
                            MC_WriteDigitalOutputErrorID_ := _AxisReference^.Data.ErrorID_AcyclicCommunication;
                            _AxisReference^.Data.CallAxisParameterMethod := TRUE;
                            _AxisReference^.Data.EnableAcyclicCommunication := FALSE;
                            THIS.AcyclicCommunicationCall(AxisRef :=  _AxisReference , DPV1ParameterNumber := TRUE, Active => Dummy);
                        ELSIF _AxisReference^.Data.CallAxisParameterMethod THEN
                            MC_WriteDigitalOutputCallNumber := MC_WriteDigitalOutputCallNumber -INT#1;
                            MC_WriteDigitalOutputDone_ := FALSE;
                            MC_WriteDigitalOutputActive_ := FALSE;
                            MC_WriteDigitalOutputError_ := TRUE;
                            MC_WriteDigitalOutputErrorID_ := AXOpen.Components.Rexroth.Drives.eAxoIndraDriveErrorCode#RESOURCE_ERROR;
                            _AxisReference^.Data.EnableAcyclicCommunication := FALSE;
                        END_IF;
                    ELSIF NOT Execute AND NOT MC_WriteDigitalOutputExecute_PV AND MC_WriteDigitalOutputCallNumber = _AxisReference^.Data.CallNumberAcyclic THEN
                        _AxisReference^.Data.CallAxisParameterMethod := TRUE;
                        _AxisReference^.Data.EnableAcyclicCommunication := FALSE;
                        THIS.AcyclicCommunicationCall(AxisRef :=  _AxisReference , DPV1ParameterNumber := TRUE, Active => Dummy);
                        MC_WriteDigitalOutputDone_ := FALSE;
                        MC_WriteDigitalOutputActive_ := FALSE;
                        MC_WriteDigitalOutputError_ := FALSE;
                        MC_WriteDigitalOutputErrorID_ := AXOpen.Components.Rexroth.Drives.eAxoIndraDriveErrorCode#NONE_ERROR;
                    ELSIF NOT Execute AND MC_WriteDigitalOutputExecute_PV THEN
                        MC_WriteDigitalOutputDone_ := FALSE;
                        MC_WriteDigitalOutputActive_ := FALSE;
                        MC_WriteDigitalOutputError_ := FALSE;
                        MC_WriteDigitalOutputErrorID_ := AXOpen.Components.Rexroth.Drives.eAxoIndraDriveErrorCode#NONE_ERROR;
                    END_IF;
                END_IF;
            END_IF;
            IF MC_WriteDigitalOutputState_ >= UINT#20 THEN
                MC_WriteDigitalOutputExecute_PV := Execute;
            END_IF;;

            Done		:= MC_WriteDigitalOutputDone_;
            Busy 		:= MC_WriteDigitalOutputActive_;
            Error 		:= MC_WriteDigitalOutputError_;
            ErrorID 	:= TO_DINT(MC_WriteDigitalOutputErrorID_);
        END_METHOD

        ///<summary>
        /// This method returns the actual position.
        ///<summary>
        METHOD PUBLIC OVERRIDE MC_ReadActualPosition
             VAR_INPUT
                AxisRef         :   AXOpen.Components.Abstractions.Drives.IAxoAxisReference;
                Enable          :   BOOL;                       //  Get the value of the parameter continuously while enabled
            END_VAR
            VAR_OUTPUT
                Valid           :   BOOL;                       //  A valid output is available at the method
                Busy            :   BOOL;                       //  The method is not finished and new output values are to be expected
                Error           :   BOOL;                       //  Signals that an error has occurred within the method
                ErrorID         :   DINT;                       //  Error identification
                Position        :   LREAL;                       //  New absolute position (in axis’ unit [u])
            END_VAR
            VAR
                _AxisReference :  REF_TO AXOpen.Components.Rexroth.Drives.AxoIndraDriveAxisReference;
                Dummy : BOOL;
            END_VAR

            _AxisReference ?= AxisRef;

            Messenger.ActivateOnCondition(ULINT#1421,_AxisReference = NULL, eAxoMessageCategory#ProgrammingError);

            IF(_AxisReference = NULL) THEN
                RETURN;
            END_IF;

            IF Enable THEN
                IF _AxisReference^.Data.CheckAccessOK	THEN
                    _AxisReference^.Data.CallAxis := TRUE;
                    _AxisReference^.Data.ReadOnlyData := TRUE;
                    THIS.FieldBusCommunication(AxisRef := _AxisReference, CommandWriteActive=> Dummy);
                    Position := _AxisReference^.Data.ActualPosition;
                    Valid := TRUE;
                    Busy := FALSE;
                    Error := FALSE;
                    ErrorID := TO_DINT(AXOpen.Components.Rexroth.Drives.eAxoIndraDriveErrorCode#NONE_ERROR);
                ELSE
                    Position := 0;
                    Error := TRUE;
                    ErrorID := TO_DINT(AXOpen.Components.Rexroth.Drives.eAxoIndraDriveErrorCode#RESOURCE_ERROR);
                END_IF;
            ELSE
                Valid := FALSE;
                Busy := FALSE;
                Error := FALSE;
                ErrorID := TO_DINT(AXOpen.Components.Rexroth.Drives.eAxoIndraDriveErrorCode#NONE_ERROR);
                Position := 0;
            END_IF;
        END_METHOD

        ///<summary>
        /// This method returns the value of the actual velocity as long as ‘Enable’ is set. ‘Valid’ is true when the
        /// dataoutput ‘Velocity’ is valid. If ‘Enable’ is Reset, the data loses its validity, and all outputs are reset,
        /// no matter if new data is available.
        ///<summary>
        METHOD PUBLIC OVERRIDE MC_ReadActualVelocity
            VAR_INPUT
                AxisRef         :   AXOpen.Components.Abstractions.Drives.IAxoAxisReference;
                Enable          :   BOOL;                       //  Get the value of the parameter continuously while enabled
            END_VAR
            VAR_OUTPUT
                Valid           :   BOOL;                       //  A valid output is available at the method
                Busy            :   BOOL;                       //  The method is not finished and new output values are to be expected
                Error           :   BOOL;                       //  Signals that an error has occurred within the method
                ErrorID         :   DINT;                       //  Error identification
                Velocity        :   LREAL;                       //  The value of the actual velocity (in axis’ unit [u/s])
            END_VAR
            VAR
                _AxisReference :  REF_TO AXOpen.Components.Rexroth.Drives.AxoIndraDriveAxisReference;
                Dummy : BOOL;
            END_VAR

            _AxisReference ?= AxisRef;

            Messenger.ActivateOnCondition(ULINT#1422,_AxisReference = NULL, eAxoMessageCategory#ProgrammingError);

            IF(_AxisReference = NULL) THEN
                RETURN;
            END_IF;

            IF Enable THEN
                IF _AxisReference^.Data.CheckAccessOK	THEN
                    _AxisReference^.Data.CallAxis := TRUE;
                    _AxisReference^.Data.ReadOnlyData := TRUE;
                    THIS.FieldBusCommunication(AxisRef:= _AxisReference,CommandWriteActive=> Dummy);
                    Velocity := _AxisReference^.Data.ActualVelocity;
                    Valid := TRUE;
                    Busy := FALSE;
                    Error := FALSE;
                    ErrorID := TO_DINT(AXOpen.Components.Rexroth.Drives.eAxoIndraDriveErrorCode#NONE_ERROR);
                ELSE
                    Velocity := 0;
                    Error := TRUE;
                    ErrorID := TO_DINT(AXOpen.Components.Rexroth.Drives.eAxoIndraDriveErrorCode#RESOURCE_ERROR);
                END_IF;
            ELSE
                Valid := FALSE;
                Busy := FALSE;
                Error := FALSE;
                ErrorID := TO_DINT(AXOpen.Components.Rexroth.Drives.eAxoIndraDriveErrorCode#NONE_ERROR);
                Velocity := 0;
            END_IF;
        END_METHOD

        ///<summary>
        /// This method returns the value of the actual torque or force as long as ‘Enable’ is set. ‘Valid’ is true when the
        /// data-output ‘Torque’ is valid. If ‘Enable’ is Reset, the data loses its validity, and ‘Valid’ is also reset,
        /// no matter if new data is available.
        ///<summary>
        METHOD PUBLIC OVERRIDE MC_ReadActualTorque
            VAR_INPUT
                AxisRef         :   AXOpen.Components.Abstractions.Drives.IAxoAxisReference;
                Enable          :   BOOL;                       //  Get the value of the parameter continuously while enabled
            END_VAR
            VAR_OUTPUT
                Valid           :   BOOL;                       //  A valid output is available at the method
                Busy            :   BOOL;                       //  The method is not finished and new output values are to be expected
                Error           :   BOOL;                       //  Signals that an error has occurred within the method
                ErrorID         :   DINT;                       //  Error identification
                Torque          :   LREAL;                       //  The value of the actual torque or force (in technical units)
            END_VAR
            VAR
                _AxisReference :  REF_TO AXOpen.Components.Rexroth.Drives.AxoIndraDriveAxisReference;
                Dummy : BOOL;
            END_VAR

            _AxisReference ?= AxisRef;

            Messenger.ActivateOnCondition(ULINT#1423,_AxisReference = NULL, eAxoMessageCategory#ProgrammingError);

            IF(_AxisReference = NULL) THEN
                RETURN;
            END_IF;

            IF Enable THEN
                IF _AxisReference^.Data.CheckAccessOK	THEN
                    _AxisReference^.Data.CallAxis := TRUE;
                    _AxisReference^.Data.ReadOnlyData := TRUE;
                    THIS.FieldBusCommunication(AxisRef:= _AxisReference,CommandWriteActive=> Dummy);
                    Torque := _AxisReference^.Data.ActualTorque;
                    Valid := TRUE;
                    Busy := FALSE;
                    Error := FALSE;
                    ErrorID := TO_DINT(AXOpen.Components.Rexroth.Drives.eAxoIndraDriveErrorCode#NONE_ERROR);
                ELSE
                    Torque := 0;
                    Error := TRUE;
                    ErrorID := TO_DINT(AXOpen.Components.Rexroth.Drives.eAxoIndraDriveErrorCode#RESOURCE_ERROR);
                END_IF;
            ELSE
                Valid := FALSE;
                Busy := FALSE;
                Error := FALSE;
                ErrorID := TO_DINT(AXOpen.Components.Rexroth.Drives.eAxoIndraDriveErrorCode#NONE_ERROR);
                Torque := 0;
            END_IF;

        END_METHOD

        ///<summary>
        /// This method returns in detail the status of the state diagram of the axis
        ///<summary>
        VAR INTERNAL
            MC_ReadStatusEnable_PV				: 	BOOL := FALSE;		//Enable - previous value
            MC_ReadStatusDone_PV				:	BOOL := FALSE;		//Done - previous value
            MC_ReadStatusStateNumber			: 	INT; 				//Call number of the method MC_ReadRealParameter
        END_VAR
        METHOD PUBLIC OVERRIDE MC_ReadStatus
            VAR_INPUT
                AxisRef         :   AXOpen.Components.Abstractions.Drives.IAxoAxisReference;
                Enable          :   BOOL;                       //  Get the value of the parameter continuously while enabled
            END_VAR
            VAR_OUTPUT
                Valid           :   BOOL;                       //  A valid output is available at the method
                Busy            :   BOOL;                       //  The method is not finished and new output values are to be expected
                Error           :   BOOL;                       //  Signals that an error has occurred within the method
                ErrorID         :   DINT;                       //  Error identification
                ErrorStop       :   BOOL;                       //  See state diagram
                Disabled        :   BOOL;                       //  See state diagram
                Stopping        :   BOOL;                       //  See state diagram
                Homing          :   BOOL;                       //  See state diagram
                Standstill      :   BOOL;                       //  See state diagram
                DiscreteMotion  :   BOOL;                       //  See state diagram
                ContinuousMotion:   BOOL;                       //  See state diagram
                SynchronizedMotion: BOOL;                       //  See state diagram
            END_VAR
            VAR
                _AxisReference :  REF_TO AXOpen.Components.Rexroth.Drives.AxoIndraDriveAxisReference;
                Dummy : BOOL;
            END_VAR

            _AxisReference ?= AxisRef;

            Messenger.ActivateOnCondition(ULINT#1424,_AxisReference = NULL, eAxoMessageCategory#ProgrammingError);

            IF(_AxisReference = NULL) THEN
                RETURN;
            END_IF;

            IF Enable THEN
                IF _AxisReference^.Data.CheckAccessOK THEN
                    Valid := TRUE;
                    Busy := FALSE;
                    _AxisReference^.Data.CallAxis := TRUE;
                    _AxisReference^.Data.ReadOnlyData := TRUE;
                    THIS.FieldBusCommunication(AxisRef:= _AxisReference,CommandWriteActive=> Dummy);
                    Errorstop := _AxisReference^.Data.StoppedDueError;
                    Stopping := _AxisReference^.Data.DriveStopReq;
                    StandStill := _AxisReference^.Data.Standstill;
                    DiscreteMotion := _AxisReference^.Data.DiscreteMotion;
                    ContinuousMotion:= _AxisReference^.Data.ContinuousMotion;
                    SynchronizedMotion := _AxisReference^.Data.SynchronizedMotion;
                    Homing := _AxisReference^.Data.HomingRunning;
                    // InPosition := _AxisReference^.Data.InPosition;
                    Error := FALSE;
                    ErrorID := TO_DINT(AXOpen.Components.Rexroth.Drives.eAxoIndraDriveErrorCode#NONE_ERROR);
                ELSE
                    Error := TRUE;
                    ErrorID := TO_DINT(AXOpen.Components.Rexroth.Drives.eAxoIndraDriveErrorCode#RESOURCE_ERROR);
                END_IF;
            ELSIF MC_ReadStatusEnable_PV THEN
                Errorstop				:= FALSE;
                Stopping				:= FALSE;
                StandStill				:= FALSE;
                DiscreteMotion		:= FALSE;
                ContinuousMotion	:= FALSE;
                SynchronizedMotion	:= FALSE;
                Homing				:= FALSE;
                // InPosition				:= FALSE;
                Valid := FALSE;
                Error := FALSE;
                ErrorID := TO_DINT(AXOpen.Components.Rexroth.Drives.eAxoIndraDriveErrorCode#NONE_ERROR);
            END_IF;
            MC_ReadStatusEnable_PV := Enable;
        END_METHOD

        ///<summary>
        /// This method returns in detail the status of the axis with respect to the motion currently in progress.
        ///<summary>
        METHOD PUBLIC OVERRIDE MC_ReadMotionState
            VAR_INPUT
                AxisRef         :   AXOpen.Components.Abstractions.Drives.IAxoAxisReference;
                Enable          :   BOOL;                       //  Get the value of the parameter continuously while enabled
                Source          :   AXOpen.Components.Abstractions.Drives.eAxoSource;                 //  Defines the source of the relevant data: CommandedValue;SetValue, ActualValue.
            END_VAR
            VAR_OUTPUT
                Valid           :   BOOL;                       //  A valid output is available at the method
                Busy            :   BOOL;                       //  The method is not finished and new output values are to be expected
                Error           :   BOOL;                       //  Signals that an error has occurred within the method
                ErrorID         :   DINT;                       //  Error identification
                ConstantVelocity:   BOOL;                       //  Velocity is constant. Velocity may be 0. For the actual value a window is applicable (window is vendor specific)
                Accelerating    :   BOOL;                       //  Increasing the absolute value of the velocity
                Decelerating    :   BOOL;                       //  Decreasing the absolute value of the velocity
                DirectionPositive:  BOOL;                       //  Signals that the position is increasing
                DirectionNegative:  BOOL;                       //  Signals that the position is decreasing
            END_VAR
            VAR
                _AxisReference :  REF_TO AXOpen.Components.Rexroth.Drives.AxoIndraDriveAxisReference;
                Dummy : BOOL;
            END_VAR

            _AxisReference ?= AxisRef;

            Messenger.ActivateOnCondition(ULINT#1425,_AxisReference = NULL, eAxoMessageCategory#ProgrammingError);

            IF(_AxisReference = NULL) THEN
                RETURN;
            END_IF;

        END_METHOD

        ///<summary>
        /// This method reads information concerning an axis, like modes, inputs directly related to the axis,
        /// and certain status information.
        ///<summary>
        METHOD PUBLIC OVERRIDE MC_ReadAxisInfo
            VAR_INPUT
                AxisRef         :   AXOpen.Components.Abstractions.Drives.IAxoAxisReference;
                Enable          :   BOOL;                       //  Get the value of the parameter continuously while enabled
            END_VAR
            VAR_OUTPUT
                Valid           :   BOOL;                       //  A valid output is available at the method
                Busy            :   BOOL;                       //  The method is not finished and new output values are to be expected
                Error           :   BOOL;                       //  Signals that an error has occurred within the method
                ErrorID         :   DINT;                       //  Error identification
                HomeAbsSwitch   :   BOOL;                       //  Digital home switch input is active
                LimitSwitchPos  :   BOOL;                       //  Positive hardware end switch is active
                LimitSwitchNeg  :   BOOL;                       //  Negative hardware end switch is active
                Simulation      :   BOOL;                       //  Axis is in simulation mode (e.g. motor is simulated)
                CommunicationReady: BOOL;                       //  “Network” is initialized and ready for communication
                ReadyForPowerOn :   BOOL;                       //  Drive is ready to be enabled (power on)
                PowerOn         :   BOOL;                       //  If TRUE shows that the power stage is switched ON
                IsHomed         :   BOOL;                       //  The absolute reference position is known for the axis (axis is homed)
                AxisWarning     :   BOOL;                       //  Warning(s) on the axis is present
            END_VAR
            VAR
                _AxisReference :  REF_TO AXOpen.Components.Rexroth.Drives.AxoIndraDriveAxisReference;
                Dummy : BOOL;
            END_VAR

            _AxisReference ?= AxisRef;

            Messenger.ActivateOnCondition(ULINT#1426,_AxisReference = NULL, eAxoMessageCategory#ProgrammingError);

            IF(_AxisReference = NULL) THEN
                RETURN;
            END_IF;

        END_METHOD

        VAR INTERNAL
            LastMessageCode :   ULINT;
        END_VAR
        ///<summary>
        /// This method presents general axis errors not relating to the methods.
        /// (for instance axis errors, drive errors, communication errors)
        ///<summary>
        METHOD PUBLIC OVERRIDE MC_ReadAxisError
            VAR_INPUT
                AxisRef         :   AXOpen.Components.Abstractions.Drives.IAxoAxisReference;
                Enable          :   BOOL;                       //  Get the value of the parameter continuously while enabled
            END_VAR
            VAR_OUTPUT
                Valid           :   BOOL;                       //  A valid output is available at the method
                Busy            :   BOOL;                       //  The method is not finished and new output values are to be expected
                Error           :   BOOL;                       //  Signals that an error has occurred within the method
                ErrorID         :   DINT;                       //  Error identification
                AxisErrorID     :   DWORD;                      //  The value of the axis error. These values are vendor specific
            END_VAR
            VAR
                _AxisReference :  REF_TO AXOpen.Components.Rexroth.Drives.AxoIndraDriveAxisReference;
                Dummy : BOOL;
                _category  :   AXOpen.Messaging.eAxoMessageCategory;
            END_VAR

            _AxisReference ?= AxisRef;

            Messenger.ActivateOnCondition(ULINT#1427,_AxisReference = NULL, eAxoMessageCategory#ProgrammingError);

            IF(_AxisReference = NULL) THEN
                RETURN;
            END_IF;

            IF Enable THEN
                IF _AxisReference^.Data.CheckAccessOK	THEN
                    _AxisReference^.Data.CallAxis := TRUE;
                    _AxisReference^.Data.ReadOnlyData := TRUE;
                    THIS.FieldBusCommunication(AxisRef := _AxisReference, CommandWriteActive=> Dummy);
                    AxisErrorID := _AxisReference^.FieldBus_In.S_0_0390_Diagnosis AND DWORD#16#000FFFFF;
                    Valid := TRUE;
                    Busy := FALSE;
                    Error := FALSE;
                    ErrorID := TO_DINT(AXOpen.Components.Rexroth.Drives.eAxoIndraDriveErrorCode#NONE_ERROR);
                    IF(AxisErrorID >= DWORD#16#000A0000 AND AxisErrorID <= DWORD#16#000AFFFF) THEN
                        _category   :=  eAxoMessageCategory#Info;
                    ELSIF(AxisErrorID >= DWORD#16#000C0000 AND AxisErrorID <= DWORD#16#000CFFFF) THEN
                        _category   :=  eAxoMessageCategory#Warning;
                    ELSIF(AxisErrorID >= DWORD#16#000E0000 AND AxisErrorID <= DWORD#16#000EFFFF) THEN
                        _category   :=  eAxoMessageCategory#Warning;
                    ELSIF(AxisErrorID >= DWORD#16#000F0000 AND AxisErrorID <= DWORD#16#000FFFFF) THEN
                        _category   :=  eAxoMessageCategory#Error;
                    END_IF;
                ELSE
                    AxisErrorID := DWORD#0;
                    Error := TRUE;
                    ErrorID := TO_DINT(AXOpen.Components.Rexroth.Drives.eAxoIndraDriveErrorCode#RESOURCE_ERROR);
                END_IF;
            ELSE
                Valid := FALSE;
                Busy := FALSE;
                Error := FALSE;
                ErrorID := TO_DINT(AXOpen.Components.Rexroth.Drives.eAxoIndraDriveErrorCode#NONE_ERROR);
                AxisErrorID := DWORD#0;
            END_IF;

            Messenger.ActivateOnCondition(LastMessageCode,Enable AND Valid AND LastMessageCode = TO_ULINT(AxisErrorID), _category);
            // IF NOT Messenger.IsActive THEN
            IF Messenger.MessengerState = eAxoMessengerState#Idle THEN
                LastMessageCode := TO_ULINT(AxisErrorID);
            END_IF;
        END_METHOD

        ///<summary>
        /// This method makes the transition from the state ‘ErrorStop’ to ‘Standstill’ or ‘Disabled’ by resetting all
        /// internal axis-related errors – it does not affect the output of the other methods.
        ///<summary>
        VAR INTERNAL
            MC_ResetExecute_PV					: 	BOOL := FALSE;		//Execute - previous value
            MC_ResetDone_PV						:	BOOL := FALSE;		//Done - previous value
            MC_ResetFirstCall					: 	BOOL;				//First call of the method MC_Reset
        END_VAR
        METHOD PUBLIC OVERRIDE MC_Reset
            VAR_INPUT
                AxisRef         :   AXOpen.Components.Abstractions.Drives.IAxoAxisReference;
                Execute         :   BOOL;                       //  Resets all internal axis-related error
            END_VAR
            VAR_OUTPUT
                Done            :   BOOL;                       //  ‘Standstill’ or ‘Disabled’ state is reached
                Busy            :   BOOL;                       //  The method is not finished and new output values are to be expected
                Error           :   BOOL;                       //  Signals that an error has occurred within the method
                ErrorID         :   DINT;                       //  Error identification
            END_VAR
            VAR
                _AxisReference :  REF_TO AXOpen.Components.Rexroth.Drives.AxoIndraDriveAxisReference;
                Dummy : BOOL;
            END_VAR

            _AxisReference ?= AxisRef;

            Messenger.ActivateOnCondition(ULINT#1428,_AxisReference = NULL, eAxoMessageCategory#ProgrammingError);

            IF(_AxisReference = NULL) THEN
                RETURN;
            END_IF;

            IF Execute THEN
                IF Execute AND NOT MC_ResetExecute_PV THEN
                    MC_ResetFirstCall := TRUE;
                    IF _AxisReference^.Data.CheckAccessOK THEN
                        Busy := TRUE;
                        _AxisReference^.Data.ResetReq := TRUE;
                    ELSE
                        Error := TRUE;
                        ErrorID := TO_DINT(AXOpen.Components.Rexroth.Drives.eAxoIndraDriveErrorCode#RESOURCE_ERROR);
                    END_IF;
                END_IF;
                IF Busy THEN
                    _AxisReference^.Data.CallAxis := TRUE;
                    _AxisReference^.Data.ReadOnlyData := FALSE;
                    Busy := TRUE;
                    THIS.FieldBusCommunication(AxisRef:= _AxisReference,CommandWriteActive=> Dummy);
                    IF  _AxisReference^.Data.ResetOK THEN
                        _AxisReference^.Data.ResetReq := FALSE;
                        Done := TRUE;
                        Busy := FALSE;
                    END_IF;
                END_IF;
            ELSIF NOT Execute AND MC_ResetExecute_PV THEN
                Done := FALSE;
                Error:=FALSE;
                ErrorID :=	TO_DINT(AXOpen.Components.Rexroth.Drives.eAxoIndraDriveErrorCode#NONE_ERROR);
                Busy := FALSE;
                IF _AxisReference^.Data.CheckAccessOK THEN
                    _AxisReference^.Data.ResetReq := FALSE;
                    _AxisReference^.Data.CallAxis := TRUE;
                    _AxisReference^.Data.ReadOnlyData := FALSE;
                    THIS.FieldBusCommunication(AxisRef:= _AxisReference,CommandWriteActive=> Dummy);
                END_IF;
            END_IF;
            IF Execute AND MC_ResetDone_PV THEN
                Done := TRUE;
            END_IF;
            MC_ResetDone_PV := Done;
            MC_ResetExecute_PV := Execute;
        END_METHOD

        METHOD PUBLIC OVERRIDE Restore
            AcyclicCommEnable_PV					:= 	FALSE;
            AcyclicCommParamNum_PV					:= 	DINT#0;
            AcyclicCommWriteValue					:= 	DINT#0;
            AcyclicCommWriteValueDW					:= 	DWORD#0;
            AcyclicCommStateCommand					:= 	INT#0;
            AcyclicCommCallNumber_PV				:=	INT#0;
            AcyclicCommDone_ 						:=	FALSE;
            AcyclicCommActive_ 						:= 	FALSE;
            AcyclicCommDecimalPlaces_ 				:=	UINT#0;
            AcyclicCommDataTypeRead_				:=	UINT#0;
            AcyclicCommDataLengthRead_				:=	UINT#0;
            AcyclicCommReadValueDINT_				:=	DINT#0;
            AcyclicCommReadValueREAL_				:=	REAL#0.0;
            AcyclicCommError_						:=	FALSE;
            AcyclicCommErrorID_						:=  eAxoIndraDriveErrorCode#NONE_ERROR;
            AcyclicCommErrorIdent_.Table            :=  AXOpen.Components.Rexroth.Drives.eAxoIndraDriveErrorTable#NO_TABLE_USED;
            AcyclicCommErrorIdent_.Additional1      :=  DWORD#0;
            AcyclicCommErrorIdent_.Additional2      :=  DWORD#0;

            CyclicCommPosition						:=	DINT#0;
            CyclicCommVelocity						:=	DINT#0;
            CyclicCommAcceleration					:=	DINT#0;
            CyclicCommDeceleration					:=	DINT#0;
            CyclicCommTorque						:=	INT#0;
            CyclicCommJerk							:=	DINT#0;
            CyclicCommVelocityWindow				:=	DINT#0;
            CyclicCommTorqueWindow					:=	INT#0;
            CyclicCommStateMachine					:=	USINT#0;
            CyclicCommSetpointAcknowledge_PV		:= 	FALSE;
            CyclicCommCheckBoundsAndMode			:= 	FALSE;
            CyclicCommWriteCommand_PV				:= 	FALSE;
            CyclicCommWaitSetpointAcknowledge		:=	FALSE;
            CyclicCommWaitSetpointReached			:= 	FALSE;
            CyclicCommCheckMultiplexDates			:= 	USINT#0;
            CyclicCommContinuousMotion				:= 	FALSE;
            CyclicCommPosVelocityWindow				:=	DINT#0;
            CyclicCommNegVelocityWindow				:=	DINT#0;
            CyclicCommPosTorqueWindow				:=	INT#0;
            CyclicCommNegTorqueWindow				:=	INT#0;
            CyclicCommActualPosition				:=	DINT#0;
            CyclicCommActualVelocity				:=  DINT#0;
            CyclicCommDiagnosis						:= 	DWORD#0;
            CyclicCommActualTorque					:=	INT#0;
            CyclicCommCommandPosition				:= 	DINT#0;
            CyclicCommCommandVelocity				:= 	DINT#1000;
            CyclicCommCommandAcceleration			:= 	DINT#1000;
            CyclicCommCommandDecceleration			:= 	DINT#1000;
            CyclicCommCommandJerk					:=	DINT#1000;
            CyclicCommCommandTorque					:= 	INT#0;
            CyclicCommMoveAdditive					:= 	FALSE;
            CyclicCommDriveStop_PV					:= 	FALSE;
            CyclicCommDriveHalt_PV					:= 	FALSE;
            CyclicCommbSelDrvOpMode3_PV				:=	FALSE;

            MC_HomeExecute_PV						:=	FALSE;
            MC_HomeCallNumber						:= 	INT#0;
            MC_HomeFirstCall						:= 	FALSE;
            MC_HomeDone_							:=	FALSE;
            MC_HomeActive_							:=	FALSE;
            MC_HomeCommandAborted_					:=	FALSE;
            MC_HomeError_							:=	FALSE;
            MC_HomeErrorID_							:=	TO_DINT(eAxoIndraDriveErrorCode#NONE_ERROR);
            MC_HomeState_							:=	UINT#0;

            MC_StopExecute_PV						:= 	FALSE;
            MC_StopCallNumber						:=	INT#0;
            MC_StopFirstCall						:= 	FALSE;

            MC_HaltExecute_PV						:= 	FALSE;
            MC_HaltCallNumber						:=	INT#0;
            MC_HaltFirstCall						:= 	FALSE;
            MC_HaltDone_							:=	FALSE;
            MC_HaltActive_							:=	FALSE;
            MC_HaltCommandAborted_					:=	FALSE;
            MC_HaltError_							:=	FALSE;
            MC_HaltErrorID_							:=	eAxoIndraDriveErrorCode#NONE_ERROR;

            MC_MoveAbsoluteExecute_PV				:= 	FALSE;
            MC_MoveAbsoluteDone_PV					:=	FALSE;
            MC_MoveAbsoluteCallNumber				:= 	INT#0;
            MC_MoveAbsoluteFirstCall				:= 	FALSE;
            MC_MoveAbsoluteDone_					:=	FALSE;
            MC_MoveAbsoluteActive_					:=	FALSE;
            MC_MoveAbsoluteCommandAborted_			:=	FALSE;
            MC_MoveAbsoluteError_					:=  FALSE;
            MC_MoveAbsoluteErrorID_					:=  eAxoIndraDriveErrorCode#NONE_ERROR;
            MC_MoveAbsoluteContinuousUpdate_PV  	:=  FALSE;

            MC_MoveRelativeExecute_PV				:= 	FALSE;
            MC_MoveRelativeDone_PV					:=	FALSE;
            MC_MoveRelativeCallNumber				:= 	INT#0;
            MC_MoveRelativeFirstCall				:= 	FALSE;
            MC_MoveRelativeDone_					:=	FALSE;
            MC_MoveRelativeActive_					:=	FALSE;
            MC_MoveRelativeCommandAborted_			:=	FALSE;
            MC_MoveRelativeError_					:=  FALSE;
            MC_MoveRelativeErrorID_					:=  eAxoIndraDriveErrorCode#NONE_ERROR;
            MC_MoveRelativeContinuousUpdate_PV  	:=  FALSE;
            MC_MoveRelativeDistance_PV          	:=  LREAL#0.0;

            MC_MoveAdditiveExecute_PV				:= 	FALSE;
            MC_MoveAdditiveDone_PV					:=	FALSE;
            MC_MoveAdditiveCallNumber				:= 	INT#0;
            MC_MoveAdditiveFirstCall				:= 	FALSE;
            MC_MoveAdditiveDone_					:=	FALSE;
            MC_MoveAdditiveActive_					:=	FALSE;
            MC_MoveAdditiveCommandAborted_			:=	FALSE;
            MC_MoveAdditiveError_					:=	FALSE;
            MC_MoveAdditiveErrorID_					:=	eAxoIndraDriveErrorCode#NONE_ERROR;
            MC_MoveAdditiveContinuousUpdate_PV  	:=  FALSE;
            MC_MoveAdditiveDistance_PV          	:=  LREAL#0.0;

            MC_MoveVelocityExecute_PV				:= 	FALSE;
            MC_MoveVelocityCallNumber				:= 	INT#0;
            MC_MoveVelocityFirstCall				:= 	FALSE;
            MC_MoveVelocityActive_					:=	FALSE;
            MC_MoveVelocityCommandAborted_			:=	FALSE;
            MC_MoveVelocityError_					:=  FALSE;
            MC_MoveVelocityErrorID_					:=  eAxoIndraDriveErrorCode#NONE_ERROR;
            MC_MoveVelocityContinuousUpdate_PV		:=  FALSE;

            MC_TorqueControlExecute_PV				:= 	FALSE;
            MC_TorqueControlCallNumber				:= 	INT#0;
            MC_TorqueControlFirstCall				:= 	FALSE;
            MC_TorqueControlActive_					:=	FALSE;
            MC_TorqueControlCommandAborted_			:=	FALSE;
            MC_TorqueControlError_					:=  FALSE;
            MC_TorqueControlErrorID_				:=  eAxoIndraDriveErrorCode#NONE_ERROR;
            MC_TorqueControlContinuousUpdate_PV 	:=  FALSE;

            MC_SetPositionDone_						:=	FALSE;
            MC_SetPositionBusy_						:=	FALSE;
            MC_SetPositionError_ 					:=	FALSE;
            MC_SetPositionErrorID_ 					:=	eAxoIndraDriveErrorCode#NONE_ERROR;
            MC_SetPositionState_ 					:=	UINT#0;
            MC_SetPositionValue_ 					:=	DINT#0;

            MC_ReadParameterEnable_PV				:= 	FALSE;
            MC_ReadParameterDone_PV					:=	FALSE;
            MC_ReadParameterCallNumber				:= 	INT#0;
            MC_ReadParameterNumber_PV				:= 	DINT#0;
            MC_ReadParameterFirstCall				:= 	FALSE;
            MC_ReadParameterDone_					:=	FALSE;
            MC_ReadParameterActive_					:=	FALSE;
            MC_ReadParameterError_					:=	FALSE;
            MC_ReadParameterErrorID_				:=	eAxoIndraDriveErrorCode#NONE_ERROR;
            MC_ReadParameterValue_					:=	DINT#0;

            MC_ReadREALParameterEnable_PV			:= 	FALSE;
            MC_ReadREALParameterDone_PV				:=	FALSE;
            MC_ReadREALParameterCallNumber			:= 	INT#0;
            MC_ReadREALParameterNumber_PV			:= 	DINT#0;
            MC_ReadREALParameterFirstCall			:= 	FALSE;
            MC_ReadREALParameterDone_				:=	FALSE;
            MC_ReadREALParameterActive_				:=	FALSE;
            MC_ReadREALParameterError_				:=	FALSE;
            MC_ReadREALParameterErrorID_			:=	eAxoIndraDriveErrorCode#NONE_ERROR;
            MC_ReadREALParameterValue_				:=	REAL#0.0;

            MC_WriteParameterExecute_PV				:= 	FALSE;
            MC_WriteParameterDone_PV				:=	FALSE;
            MC_WriteParameterCallNumber				:= 	DINT#0;
            MC_WriteParameterFirstCall				:= 	FALSE;
            MC_WriteParameterDone_					:=	FALSE;
            MC_WriteParameterActive_				:=	FALSE;
            MC_WriteParameterError_					:=	FALSE;
            MC_WriteParameterErrorID_				:=	eAxoIndraDriveErrorCode#NONE_ERROR;

            MC_WriteREALParameterExecute_PV			:= 	FALSE;
            MC_WriteREALParameterDone_PV			:=	FALSE;
            MC_WriteREALParameterCallNumber			:= 	INT#0;
            MC_WriteREALParameterFirstCall			:= 	FALSE;
            MC_WriteREALParameterDone_				:=	FALSE;
            MC_WriteREALParameterActive_			:=	FALSE;
            MC_WriteREALParameterError_				:=	FALSE;
            MC_WriteREALParameterErrorID_			:=	eAxoIndraDriveErrorCode#NONE_ERROR;

            MC_ReadDigitalInputEnable_PV			:= 	FALSE;
            MC_ReadDigitalInputDone_PV				:=	FALSE;
            MC_ReadDigitalInputCallNumber			:= 	INT#0;
            MC_ReadDigitalInputNumber_PV			:= 	DINT#0;
            MC_ReadDigitalInputFirstCall			:= 	FALSE;
            MC_ReadDigitalInputDone_				:=	FALSE;
            MC_ReadDigitalInputActive_				:=	FALSE;
            MC_ReadDigitalInputError_				:=	FALSE;
            MC_ReadDigitalInputErrorID_				:=	eAxoIndraDriveErrorCode#NONE_ERROR;
            MC_ReadDigitalInputValue_				:=	DINT#0;

            MC_ReadDigitalOutputEnable_PV			:= 	FALSE;
            MC_ReadDigitalOutputDone_PV				:=	FALSE;
            MC_ReadDigitalOutputCallNumber			:= 	INT#0;
            MC_ReadDigitalOutputNumber_PV			:= 	DINT#0;
            MC_ReadDigitalOutputFirstCall			:= 	FALSE;
            MC_ReadDigitalOutputDone_				:=	FALSE;
            MC_ReadDigitalOutputActive_				:=	FALSE;
            MC_ReadDigitalOutputError_				:=	FALSE;
            MC_ReadDigitalOutputErrorID_			:=	eAxoIndraDriveErrorCode#NONE_ERROR;
            MC_ReadDigitalOutputValue_				:=	DINT#0;

            MC_WriteDigitalOutputExecute_PV			:= 	FALSE;
            MC_WriteDigitalOutputDone_PV			:=	FALSE;
            MC_WriteDigitalOutputCallNumber			:= 	INT#0;
            MC_WriteDigitalOutputFirstCall			:= 	FALSE;
            MC_WriteDigitalOutputDone_				:=	FALSE;
            MC_WriteDigitalOutputActive_			:=	FALSE;
            MC_WriteDigitalOutputError_				:=	FALSE;
            MC_WriteDigitalOutputErrorID_			:=	eAxoIndraDriveErrorCode#NONE_ERROR;
            MC_WriteDigitalOutputState_				:=	UINT#0;
            MC_WriteDigitalOutputValueRead_ 		:=	LINT#0;
            MC_WriteDigitalOutputValueToWrite_		:=	LINT#0;

            MC_ReadStatusEnable_PV					:= 	FALSE;
            MC_ReadStatusDone_PV					:=	FALSE;
            MC_ReadStatusStateNumber				:= 	INT#0;

            LastMessageCode :=   ULINT#0;

            MC_ResetExecute_PV						:= 	FALSE;
            MC_ResetDone_PV							:=	FALSE;
            MC_ResetFirstCall						:= 	FALSE;

            DriveStatus.Action.Id := UINT#0;
            DriveStatus.Error.Id  := UINT#0;
            Messenger.Restore();
            TaskMessenger.Restore();

            //AxoPower_Task.Restore();
            AxoStop_Task.Restore();
            AxoHalt_Task.Restore();
            AxoHome_Task.Restore();
            AxoMoveAbsolute_Task.Restore();
            AxoMoveRelative_Task.Restore();
            AxoMoveAdditive_Task.Restore();
            AxoMoveVelocity_Task.Restore();
            AxoTorqueControl_Task.Restore();
            AxoSetPosition_Task.Restore();
            AxoSetOverride_Task.SwitchOff();
            AxoReadParameter_Task.SwitchOff();
            AxoReadRealParameter_Task.SwitchOff();
            AxoReadBoolParameter_Task.SwitchOff();
            AxoWriteParameter_Task.Restore();
            AxoWriteRealParameter_Task.Restore();
            AxoWriteBoolParameter_Task.Restore();
            AxoReadDigitalInput_Task.SwitchOff();
            AxoReadDigitalOutput_Task.SwitchOff();
            AxoWriteDigitalOutput_Task.Restore();
            AxoReadActualPosition_Task.SwitchOff();
            AxoReadActualVelocity_Task.SwitchOff();
            AxoReadActualTorque_Task.SwitchOff();
            AxoReadStatus_Task.SwitchOff();
            AxoReadMotionState_Task.SwitchOff();
            AxoReadAxisInfo_Task.SwitchOff();
            AxoReadAxisError_Task.SwitchOff();
            AxoReset_Task.Restore();
            AxoJogPositive.RemoteSwitchOn := FALSE;
            AxoJogPositive.StartMotion := FALSE;
            AxoJogPositive.StopMotion := FALSE;
            AxoJogNegative.RemoteSwitchOn := FALSE;
            AxoJogNegative.StartMotion := FALSE;
            AxoJogNegative.StopMotion := FALSE;

            RestoreTask.DoneWhen(TRUE);
            SUPER.Restore();
        END_METHOD
    END_CLASS
END_NAMESPACE
